//{attribute 'qualified_only'}
VAR_GLOBAL
	
//Example implementation of the FFO
    {attribute 'pytmc' := '
    pv: PLC:LFE:VAC:FF1
    '}
    {attribute 'TcLinkTo' := '.q_xFastFaultOut:=TIIB[PLC_E1_EL2202]^Channel 1^Output'}
    g_FastFaultOutput1  :   FB_HardwareFFOutput;	//FFO for ST1L0_XTES's Upstream Components
	
	 {attribute 'pytmc' := '
    pv: PLC:LFE:VAC:FF2
    '}
    {attribute 'TcLinkTo' := '.q_xFastFaultOut:=TIIB[PLC_E1_EL2202]^Channel 2^Output'}
    g_FastFaultOutput2  :   FB_HardwareFFOutput;	//FFO for ST1L0_XTES's Downstream Components
	
	{attribute 'pytmc' := '
    pv: PLC:LFE:VAC:RESET:FF1
    '}
	xReset_PMPS_FFO1	:	BOOL	:=	FALSE;		//FFO RESET for ST1L0_XTES's Upstream Components
	{attribute 'pytmc' := '
    pv: PLC:LFE:VAC:RESET:FF2
    '}
	xReset_PMPS_FFO2	:	BOOL	:=	FALSE;		//FFO RESET for ST1L0_XTES's Downstream Components
	
	
	xEBD_FEE_MPS_OK: BOOL := TRUE;
	xH1_1_H1_2_MPS_OK: BOOL;

END_VAR

(* stored: Version 1.1.0.1, ProductVersion 3.1.4022.12
   GVL GVL_PMPS: Id {4625b23c-c93c-4b67-8375-0fbf2be37f8b} *)
